INTERFACE I_BoolPub EXTENDS I_SYS_COMP_Object

METHOD Attach_Sub
VAR_INPUT
	IObject: I_SYS_COMP_Object;
END_VAR
END_METHOD

PROPERTY Get : BOOL
GET
END_GET
END_PROPERTY

METHOD Remove_Sub
VAR_INPUT
	IObject: I_SYS_COMP_Object;
END_VAR
END_METHOD

END_INTERFACE

(* stored: Version 1.1.0.1, ProductVersion 3.1.4024.12
   Itf I_BoolPub: Id {0c8aefb5-64be-4ef0-bee9-a126844e4796}
   Method Attach_Sub: Id {69b208be-e7fc-426f-bdc1-fee6bcdf39b6}
   Property Get: Id {c5490e48-569b-4dc5-b268-e6b049cc851f}
   Get Get: Id {af43da6a-d8ed-4372-885e-188bc70ed501}
   Method Remove_Sub: Id {2a04d141-1a4d-4e1e-acb1-2a9e369ae058} *)
